// Mitsubishi GX Works2 project: a1   PLC: Q02/Q02H

PROGRAM MAIN
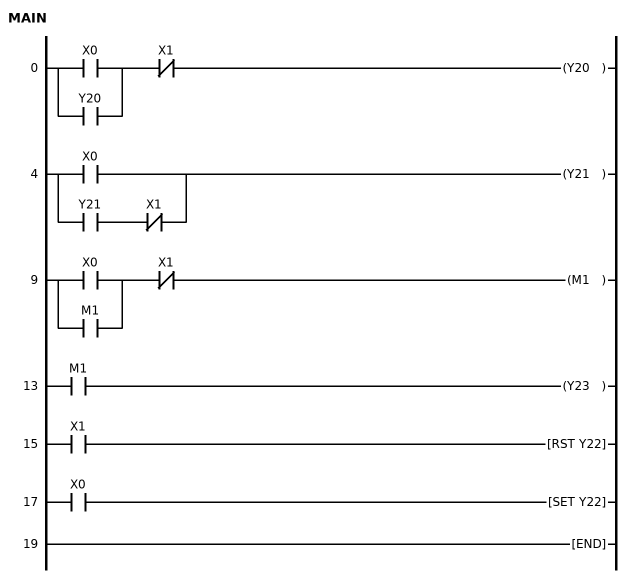
0     LD      X0
      OR      Y20
      ANI     X1
      OUT     Y20
4     LD      X0
      LD      Y21
      ANI     X1
      ORB
      OUT     Y21
9     LD      X0
      OR      M1
      ANI     X1
      OUT     M1
13    LD      M1
      OUT     Y23
15    LD      X1
      RST     Y22
17    LD      X0
      SET     Y22
19    END
END_PROGRAM
